// TIA Portal V21 export
FUNCTION_BLOCK "FB304"   // FB304, LAD
TITLE = FB304
{ S7_Optimized_Access := 'TRUE' }
AUTHOR : PRECISE
FAMILY : PRECISE
// BLANKETING
// stored: AutoNumber false, MemoryReserve 100, SetENOAutomatically false
   VAR_INPUT
      Enable : Bool;
      Disable : Bool;
      Fault : Bool;
      SecPulse : Bool;
      AlwaysTrue : Bool;
      StartConfirmationPopupSel : Bool;   // StartConfirmationPopupSel: 0-NO/1-YES
      EndConfirmationPopupSel : Bool;   // EndConfirmationPopupSel: 0-NO/1-YES
      BlanketingModeSel : Int;   // Blanketing Mode Selection: 0-Pressure/1-Pressure+Time
      BlanketingTimebaseSel : Bool;   // Blanketing Timebase Selection: 0-sec/1-min
      GasSel : Int;   // Gas Selection - 0-AIR/1-N2
      SetPressure : Real := 1.0;   // For Blanketing Mode Selection: 0-Pressure
      BlanketingTimeMin : Int := 1;   // For Blanketing Mode Selection: 1-Pressure+Time & Blanketing Timebase Selection: 1-min
      BlanketingTimeSec : Int := 30;   // For Blanketing Mode Selection: 1-Pressure+Time & Blanketing Timebase Selection: 0-sec
      ActualPressure : Real;   // For Sparging LineSelection: 1-THRU VV
      DelaytoOpenGasIn : Int := 3;
      PressureTol : Real := 0.3;
   END_VAR
   VAR_OUTPUT
      AirValve : Bool;
      N2Valve : Bool;
      BlanketingLineValves : Bool;
      StartConfirmationPopup : Bool;   // For Start Confirmation Popup Selection: Yes
      EndConfirmationPopup : Bool;   // For End Confirmation Popup Selection: Yes
      BlanketingTimeMinPV : DInt;
      BlanketingTimeSecPV : DInt;
      PrintTrigger : Bool;
      PrintWord : Int;
      PrintStatus : String[50];
   END_VAR
   VAR_IN_OUT
      Start : Bool;
      Stop : Bool;
      Reset : Bool;
      StartConfirmationAck : Bool;   // For Start Confirmation Popup Selection: Yes
      EndConfirmationAck : Bool;   // For End Confirmation Popup Selection: Yes
      SpareBtn1 : Bool;
      SpareBtn2 : Bool;
      SpareBtn3 : Bool;
      Running : Bool;
      Selected : Bool;
      Paused : Bool;
      StartConfirmationPopupTemp : Bool;   // For Start Confirmation Popup Selection: Yes
      EndConfirmationPopupTemp : Bool;   // For End Confirmation Popup Selection: Yes
      BlanketingStarted : Bool;
      BlanketingOver : Bool;
      BlanketingTimerRunning : Bool;
      PressureTolNeg : Real;
   END_VAR
   VAR
      ValveOnDelayPV : Int;
      ValveOffDelayPV : Int;
      PrintTriggerTemp : Bool;
      RE1 : Bool;
      RE2 : Bool;
      RE3 : Bool;
      RE4 : Bool;
      RE5 : Bool;
      RE6 : Bool;
      RE7 : Bool;
      BlanketingTimer { S7_SetPoint := 'True'} : "FB101";
      PrintTriggerResetTimer { S7_SetPoint := 'True'} : TON_TIME;
      BtnResetTimer { S7_SetPoint := 'True'} : TON_TIME;
   END_VAR
   VAR_TEMP
      STATUS1 : String[40];
      STATUS2 : String[40];
      STATUS3 : String[40];
      STATUS4 : String[40];
      STATUS5 : String[40];
   END_VAR
   VAR_TEMP   // added for the SCL form of the ladder/FBD networks
      _w1 : Bool;
      _w2 : Bool;
      _w3 : Bool;
      _w4 : Bool;
      _w5 : Bool;
   END_VAR
BEGIN

REGION Network 1: Running
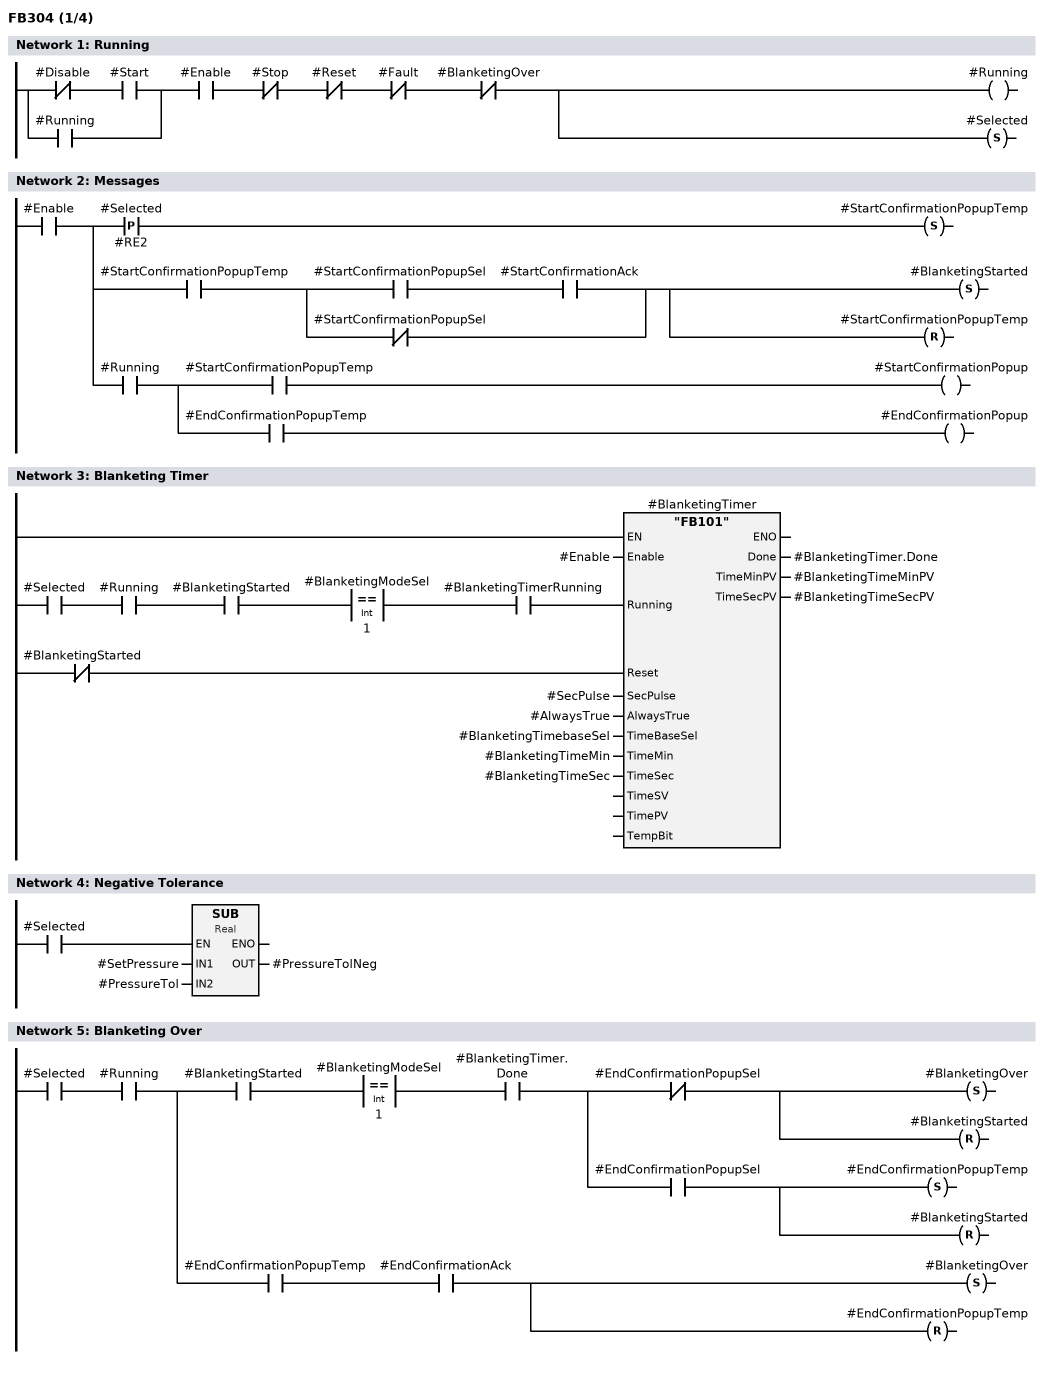
   RUNG wire#powerrail
      I_Contact( #Disable )
      Contact( #Start )
      wire#w1
      Contact( #Enable )
      I_Contact( #Stop )
      I_Contact( #Reset )
      I_Contact( #Fault )
      I_Contact( #BlanketingOver )
      wire#w2
      Coil( #Running )
   END_RUNG
   RUNG wire#powerrail
      Contact( #Running )
   END_RUNG wire#w1
   RUNG wire#w2
      S_Coil( #Selected )
   END_RUNG
   // the same network as SCL:
   #Running := ((NOT #Disable AND #Start) OR #Running) AND #Enable AND NOT #Stop AND NOT #Reset AND NOT #Fault AND NOT #BlanketingOver;
   IF #Running THEN #Selected := TRUE; END_IF;
END_REGION

REGION Network 2: Messages
   RUNG wire#powerrail
      Contact( #Enable )
      wire#w1
      P_Contact(operand := #Selected, bit := #RE2)
      S_Coil( #StartConfirmationPopupTemp )
   END_RUNG
   RUNG wire#w1
      Contact( #StartConfirmationPopupTemp )
      wire#w2
      Contact( #StartConfirmationPopupSel )
      Contact( #StartConfirmationAck )
      wire#w3
      S_Coil( #BlanketingStarted )
   END_RUNG
   RUNG wire#w2
      I_Contact( #StartConfirmationPopupSel )
   END_RUNG wire#w3
   RUNG wire#w3
      R_Coil( #StartConfirmationPopupTemp )
   END_RUNG
   RUNG wire#w1
      Contact( #Running )
      wire#w4
      Contact( #StartConfirmationPopupTemp )
      Coil( #StartConfirmationPopup )
   END_RUNG
   RUNG wire#w4
      Contact( #EndConfirmationPopupTemp )
      Coil( #EndConfirmationPopup )
   END_RUNG
   // the same network as SCL:
   #_w1 := #Enable AND #Selected AND NOT #RE2;   // rising edge of #Selected
   #RE2 := #Selected;
   IF #_w1 THEN #StartConfirmationPopupTemp := TRUE; END_IF;
   IF #Enable AND #StartConfirmationPopupTemp AND ((#StartConfirmationPopupSel AND #StartConfirmationAck) OR NOT #StartConfirmationPopupSel) THEN
       #BlanketingStarted := TRUE;
       #StartConfirmationPopupTemp := FALSE;
   END_IF;
   #_w2 := #Enable AND #Running;
   #StartConfirmationPopup := #_w2 AND #StartConfirmationPopupTemp;
   #EndConfirmationPopup := #_w2 AND #EndConfirmationPopupTemp;
END_REGION

REGION Network 3: Blanketing Timer
   RUNG wire#powerrail
      #BlanketingTimer(Running := wire#w1, Reset := wire#w2, Enable := #Enable, SecPulse := #SecPulse, AlwaysTrue := #AlwaysTrue, TimeBaseSel := #BlanketingTimebaseSel, TimeMin := #BlanketingTimeMin, TimeSec := #BlanketingTimeSec, TimeSV :=, TimePV :=, TempBit :=, Done => #BlanketingTimer.Done, TimeMinPV => #BlanketingTimeMinPV, TimeSecPV => #BlanketingTimeSecPV)
   END_RUNG
   RUNG wire#powerrail
      Contact( #Selected )
      Contact( #Running )
      Contact( #BlanketingStarted )
      { S7_Templates := "SrcType := Int" } EQ_Contact(in1 := #BlanketingModeSel, in2 := 1)
      Contact( #BlanketingTimerRunning )
   END_RUNG wire#w1
   RUNG wire#powerrail
      I_Contact( #BlanketingStarted )
   END_RUNG wire#w2
   // the same network as SCL:
   #BlanketingTimer(Enable := #Enable,   // "FB101"
                    Running := #Selected AND #Running AND #BlanketingStarted AND (#BlanketingModeSel = 1) AND #BlanketingTimerRunning,
                    Reset := NOT #BlanketingStarted,
                    SecPulse := #SecPulse,
                    AlwaysTrue := #AlwaysTrue,
                    TimeBaseSel := #BlanketingTimebaseSel,
                    TimeMin := #BlanketingTimeMin,
                    TimeSec := #BlanketingTimeSec,
                    Done => #BlanketingTimer.Done,
                    TimeMinPV => #BlanketingTimeMinPV,
                    TimeSecPV => #BlanketingTimeSecPV);
END_REGION

REGION Network 4: Negative Tolerance
   RUNG wire#powerrail
      Contact( #Selected )
      { S7_Templates := "SrcType := Real"; S7_GenerateENO := "TRUE" } Sub(in1 := #SetPressure, in2 := #PressureTol, out => #PressureTolNeg)
   END_RUNG
   // the same network as SCL:
   IF #Selected THEN #PressureTolNeg := #SetPressure - #PressureTol; END_IF;
END_REGION

REGION Network 5: Blanketing Over
   RUNG wire#powerrail
      Contact( #Selected )
      Contact( #Running )
      wire#w1
      Contact( #BlanketingStarted )
      { S7_Templates := "SrcType := Int" } EQ_Contact(in1 := #BlanketingModeSel, in2 := 1)
      Contact( #BlanketingTimer.Done )
      wire#w2
      I_Contact( #EndConfirmationPopupSel )
      wire#w3
      S_Coil( #BlanketingOver )
   END_RUNG
   RUNG wire#w3
      R_Coil( #BlanketingStarted )
   END_RUNG
   RUNG wire#w2
      Contact( #EndConfirmationPopupSel )
      wire#w4
      S_Coil( #EndConfirmationPopupTemp )
   END_RUNG
   RUNG wire#w4
      R_Coil( #BlanketingStarted )
   END_RUNG
   RUNG wire#w1
      Contact( #EndConfirmationPopupTemp )
      Contact( #EndConfirmationAck )
      wire#w5
      S_Coil( #BlanketingOver )
   END_RUNG
   RUNG wire#w5
      R_Coil( #EndConfirmationPopupTemp )
   END_RUNG
   // the same network as SCL:
   #_w1 := #Selected AND #Running;
   #_w2 := #_w1 AND #BlanketingStarted AND (#BlanketingModeSel = 1) AND #BlanketingTimer.Done;
   IF #_w2 AND NOT #EndConfirmationPopupSel THEN
       #BlanketingOver := TRUE;
       #BlanketingStarted := FALSE;
   END_IF;
   IF #_w2 AND #EndConfirmationPopupSel THEN
       #EndConfirmationPopupTemp := TRUE;
       #BlanketingStarted := FALSE;
   END_IF;
   IF #_w1 AND #EndConfirmationPopupTemp AND #EndConfirmationAck THEN
       #BlanketingOver := TRUE;
       #EndConfirmationPopupTemp := FALSE;
   END_IF;
END_REGION

REGION Network 6: Output On
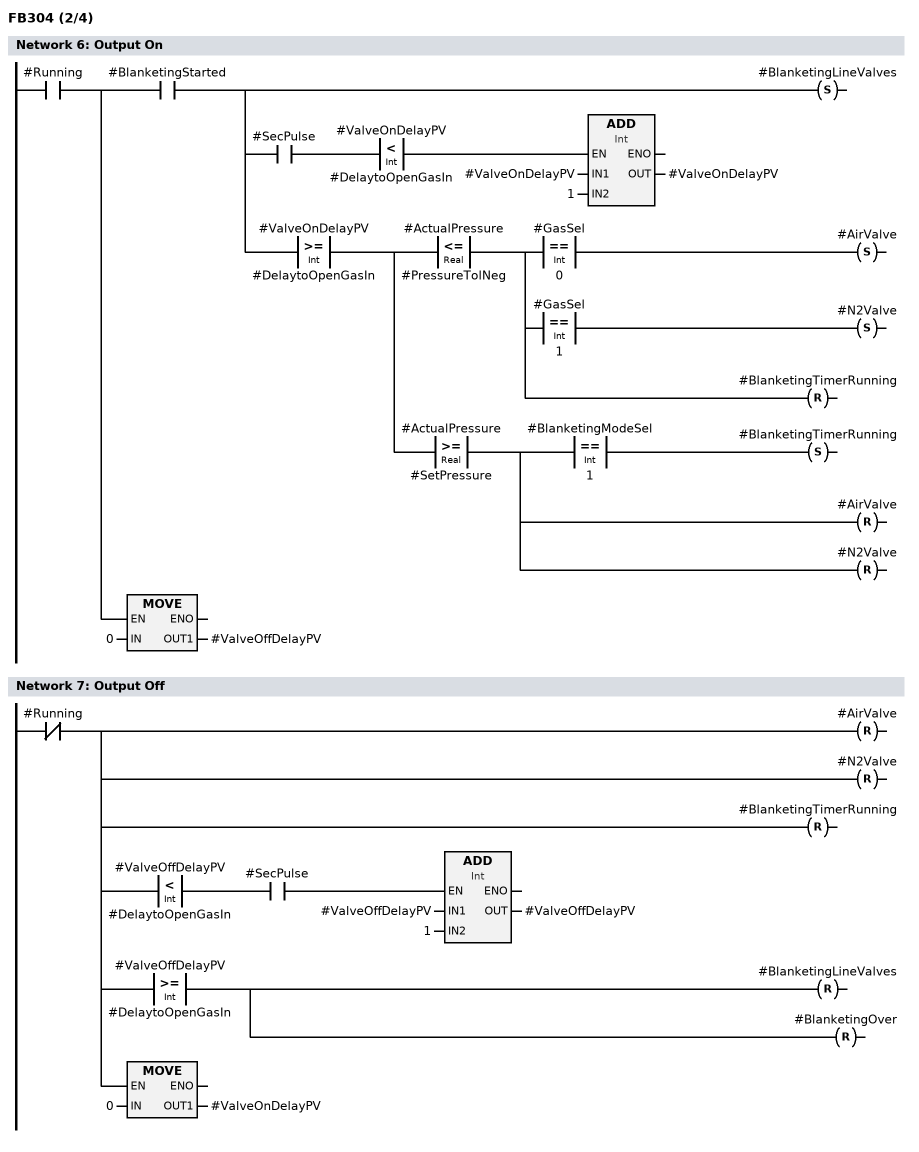
   RUNG wire#powerrail
      Contact( #Running )
      wire#w1
      Contact( #BlanketingStarted )
      wire#w2
      S_Coil( #BlanketingLineValves )
   END_RUNG
   RUNG wire#w2
      Contact( #SecPulse )
      { S7_Templates := "SrcType := Int" } LT_Contact(in1 := #ValveOnDelayPV, in2 := #DelaytoOpenGasIn)
      { S7_Templates := "SrcType := Int"; S7_GenerateENO := "TRUE" } Add(in1 := #ValveOnDelayPV, in2 := 1, out => #ValveOnDelayPV)
   END_RUNG
   RUNG wire#w2
      { S7_Templates := "SrcType := Int" } GE_Contact(in1 := #ValveOnDelayPV, in2 := #DelaytoOpenGasIn)
      wire#w3
      { S7_Templates := "SrcType := Real" } LE_Contact(in1 := #ActualPressure, in2 := #PressureTolNeg)
      wire#w4
      { S7_Templates := "SrcType := Int" } EQ_Contact(in1 := #GasSel, in2 := 0)
      S_Coil( #AirValve )
   END_RUNG
   RUNG wire#w4
      { S7_Templates := "SrcType := Int" } EQ_Contact(in1 := #GasSel, in2 := 1)
      S_Coil( #N2Valve )
   END_RUNG
   RUNG wire#w4
      R_Coil( #BlanketingTimerRunning )
   END_RUNG
   RUNG wire#w3
      { S7_Templates := "SrcType := Real" } GE_Contact(in1 := #ActualPressure, in2 := #SetPressure)
      wire#w5
      { S7_Templates := "SrcType := Int" } EQ_Contact(in1 := #BlanketingModeSel, in2 := 1)
      S_Coil( #BlanketingTimerRunning )
   END_RUNG
   RUNG wire#w5
      R_Coil( #AirValve )
   END_RUNG
   RUNG wire#w5
      R_Coil( #N2Valve )
   END_RUNG
   RUNG wire#w1
      { S7_GenerateENO := "TRUE" } Move(in := 0, out1 => #ValveOffDelayPV)
   END_RUNG
   // the same network as SCL:
   #_w1 := #Running AND #BlanketingStarted;
   IF #_w1 THEN #BlanketingLineValves := TRUE; END_IF;
   IF #_w1 AND #SecPulse AND (#ValveOnDelayPV < #DelaytoOpenGasIn) THEN
       #ValveOnDelayPV := #ValveOnDelayPV + 1;
   END_IF;
   #_w2 := #_w1 AND (#ValveOnDelayPV >= #DelaytoOpenGasIn);
   #_w3 := #_w2 AND (#ActualPressure <= #PressureTolNeg);
   IF #_w3 AND (#GasSel = 0) THEN #AirValve := TRUE; END_IF;
   IF #_w3 AND (#GasSel = 1) THEN #N2Valve := TRUE; END_IF;
   IF #_w3 THEN #BlanketingTimerRunning := FALSE; END_IF;
   #_w4 := #_w2 AND (#ActualPressure >= #SetPressure);
   IF #_w4 AND (#BlanketingModeSel = 1) THEN #BlanketingTimerRunning := TRUE; END_IF;
   IF #_w4 THEN
       #AirValve := FALSE;
       #N2Valve := FALSE;
   END_IF;
   IF #Running THEN #ValveOffDelayPV := 0; END_IF;
END_REGION

REGION Network 7: Output Off
   RUNG wire#powerrail
      I_Contact( #Running )
      wire#w1
      R_Coil( #AirValve )
   END_RUNG
   RUNG wire#w1
      R_Coil( #N2Valve )
   END_RUNG
   RUNG wire#w1
      R_Coil( #BlanketingTimerRunning )
   END_RUNG
   RUNG wire#w1
      { S7_Templates := "SrcType := Int" } LT_Contact(in1 := #ValveOffDelayPV, in2 := #DelaytoOpenGasIn)
      Contact( #SecPulse )
      { S7_Templates := "SrcType := Int"; S7_GenerateENO := "TRUE" } Add(in1 := #ValveOffDelayPV, in2 := 1, out => #ValveOffDelayPV)
   END_RUNG
   RUNG wire#w1
      { S7_Templates := "SrcType := Int" } GE_Contact(in1 := #ValveOffDelayPV, in2 := #DelaytoOpenGasIn)
      wire#w2
      R_Coil( #BlanketingLineValves )
   END_RUNG
   RUNG wire#w2
      R_Coil( #BlanketingOver )
   END_RUNG
   RUNG wire#w1
      { S7_GenerateENO := "TRUE" } Move(in := 0, out1 => #ValveOnDelayPV)
   END_RUNG
   // the same network as SCL:
   IF NOT #Running THEN
       #AirValve := FALSE;
       #N2Valve := FALSE;
       #BlanketingTimerRunning := FALSE;
   END_IF;
   IF NOT #Running AND (#ValveOffDelayPV < #DelaytoOpenGasIn) AND #SecPulse THEN
       #ValveOffDelayPV := #ValveOffDelayPV + 1;
   END_IF;
   IF NOT #Running AND (#ValveOffDelayPV >= #DelaytoOpenGasIn) THEN
       #BlanketingLineValves := FALSE;
       #BlanketingOver := FALSE;
   END_IF;
   IF NOT #Running THEN #ValveOnDelayPV := 0; END_IF;
END_REGION

REGION Network 8: Event Status
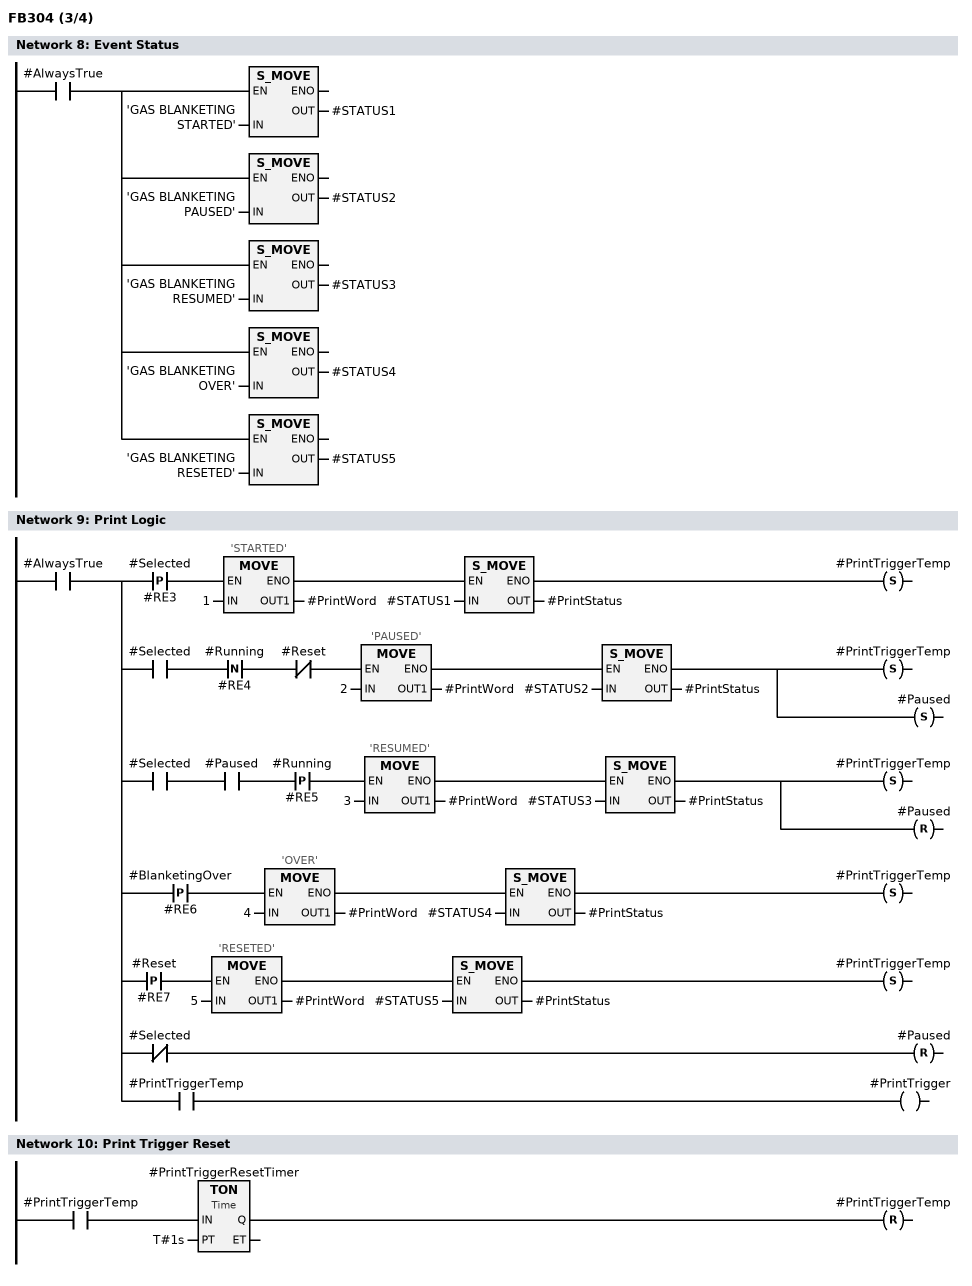
   RUNG wire#powerrail
      Contact( #AlwaysTrue )
      wire#w1
      S_Move(in := 'GAS BLANKETING STARTED', out => #STATUS1)
   END_RUNG
   RUNG wire#w1
      S_Move(in := 'GAS BLANKETING PAUSED', out => #STATUS2)
   END_RUNG
   RUNG wire#w1
      S_Move(in := 'GAS BLANKETING RESUMED', out => #STATUS3)
   END_RUNG
   RUNG wire#w1
      S_Move(in := 'GAS BLANKETING OVER', out => #STATUS4)
   END_RUNG
   RUNG wire#w1
      S_Move(in := 'GAS BLANKETING RESETED', out => #STATUS5)
   END_RUNG
   // the same network as SCL:
   IF #AlwaysTrue THEN
       #STATUS1 := 'GAS BLANKETING STARTED';
       #STATUS2 := 'GAS BLANKETING PAUSED';
       #STATUS3 := 'GAS BLANKETING RESUMED';
       #STATUS4 := 'GAS BLANKETING OVER';
       #STATUS5 := 'GAS BLANKETING RESETED';
   END_IF;
END_REGION

REGION Network 9: Print Logic
   RUNG wire#powerrail
      Contact( #AlwaysTrue )
      wire#w1
      P_Contact(operand := #Selected, bit := #RE3)
      { S7_GenerateENO := "TRUE" } Move(in := 1, out1 => #PrintWord)   // 'STARTED'
      S_Move(in := #STATUS1, out => #PrintStatus)
      S_Coil( #PrintTriggerTemp )
   END_RUNG
   RUNG wire#w1
      Contact( #Selected )
      N_Contact(operand := #Running, bit := #RE4)
      I_Contact( #Reset )
      { S7_GenerateENO := "TRUE" } Move(in := 2, out1 => #PrintWord)   // 'PAUSED'
      S_Move(in := #STATUS2, out => #PrintStatus)
      wire#w2
      S_Coil( #PrintTriggerTemp )
   END_RUNG
   RUNG wire#w2
      S_Coil( #Paused )
   END_RUNG
   RUNG wire#w1
      Contact( #Selected )
      Contact( #Paused )
      P_Contact(operand := #Running, bit := #RE5)
      { S7_GenerateENO := "TRUE" } Move(in := 3, out1 => #PrintWord)   // 'RESUMED'
      S_Move(in := #STATUS3, out => #PrintStatus)
      wire#w3
      S_Coil( #PrintTriggerTemp )
   END_RUNG
   RUNG wire#w3
      R_Coil( #Paused )
   END_RUNG
   RUNG wire#w1
      P_Contact(operand := #BlanketingOver, bit := #RE6)
      { S7_GenerateENO := "TRUE" } Move(in := 4, out1 => #PrintWord)   // 'OVER'
      S_Move(in := #STATUS4, out => #PrintStatus)
      S_Coil( #PrintTriggerTemp )
   END_RUNG
   RUNG wire#w1
      P_Contact(operand := #Reset, bit := #RE7)
      { S7_GenerateENO := "TRUE" } Move(in := 5, out1 => #PrintWord)   // 'RESETED'
      S_Move(in := #STATUS5, out => #PrintStatus)
      S_Coil( #PrintTriggerTemp )
   END_RUNG
   RUNG wire#w1
      I_Contact( #Selected )
      R_Coil( #Paused )
   END_RUNG
   RUNG wire#w1
      Contact( #PrintTriggerTemp )
      Coil( #PrintTrigger )
   END_RUNG
   // the same network as SCL:
   // ENO of a box is taken as its EN; it also drops when the box reports an error
   #_w1 := #AlwaysTrue AND #Selected AND NOT #RE3;   // rising edge of #Selected
   #RE3 := #Selected;
   IF #_w1 THEN
       #PrintWord := 1;   // 'STARTED'
       #PrintStatus := #STATUS1;
       #PrintTriggerTemp := TRUE;
   END_IF;
   #_w2 := #AlwaysTrue AND #Selected AND NOT #Running AND #RE4;   // falling edge of #Running
   #RE4 := #Running;
   IF #_w2 AND NOT #Reset THEN
       #PrintWord := 2;   // 'PAUSED'
       #PrintStatus := #STATUS2;
       #PrintTriggerTemp := TRUE;
       #Paused := TRUE;
   END_IF;
   #_w3 := #AlwaysTrue AND #Selected AND #Paused AND #Running AND NOT #RE5;   // rising edge of #Running
   #RE5 := #Running;
   IF #_w3 THEN
       #PrintWord := 3;   // 'RESUMED'
       #PrintStatus := #STATUS3;
       #PrintTriggerTemp := TRUE;
       #Paused := FALSE;
   END_IF;
   #_w4 := #AlwaysTrue AND #BlanketingOver AND NOT #RE6;   // rising edge of #BlanketingOver
   #RE6 := #BlanketingOver;
   IF #_w4 THEN
       #PrintWord := 4;   // 'OVER'
       #PrintStatus := #STATUS4;
       #PrintTriggerTemp := TRUE;
   END_IF;
   #_w5 := #AlwaysTrue AND #Reset AND NOT #RE7;   // rising edge of #Reset
   #RE7 := #Reset;
   IF #_w5 THEN
       #PrintWord := 5;   // 'RESETED'
       #PrintStatus := #STATUS5;
       #PrintTriggerTemp := TRUE;
   END_IF;
   IF #AlwaysTrue AND NOT #Selected THEN #Paused := FALSE; END_IF;
   #PrintTrigger := #AlwaysTrue AND #PrintTriggerTemp;
END_REGION

REGION Network 10: Print Trigger Reset
   RUNG wire#powerrail
      Contact( #PrintTriggerTemp )
      { S7_Templates := "time_type := Time" } #PrintTriggerResetTimer.TON(pt := T#1s, et =>)
      R_Coil( #PrintTriggerTemp )
   END_RUNG
   // the same network as SCL:
   #PrintTriggerResetTimer(IN := #PrintTriggerTemp, PT := T#1s);   // TON
   IF #PrintTriggerResetTimer.Q THEN #PrintTriggerTemp := FALSE; END_IF;
END_REGION

REGION Network 11: Button Reset
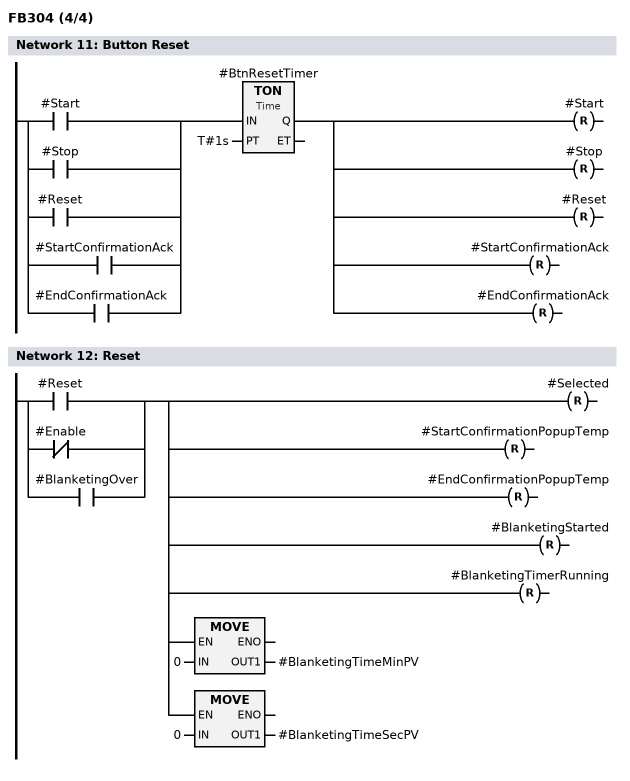
   RUNG wire#powerrail
      Contact( #Start )
      wire#w1
      { S7_Templates := "time_type := Time" } #BtnResetTimer.TON(pt := T#1s, et =>)
      wire#w2
      R_Coil( #Start )
   END_RUNG
   RUNG wire#powerrail
      Contact( #Stop )
   END_RUNG wire#w1
   RUNG wire#powerrail
      Contact( #Reset )
   END_RUNG wire#w1
   RUNG wire#powerrail
      Contact( #StartConfirmationAck )
   END_RUNG wire#w1
   RUNG wire#powerrail
      Contact( #EndConfirmationAck )
   END_RUNG wire#w1
   RUNG wire#w2
      R_Coil( #Stop )
   END_RUNG
   RUNG wire#w2
      R_Coil( #Reset )
   END_RUNG
   RUNG wire#w2
      R_Coil( #StartConfirmationAck )
   END_RUNG
   RUNG wire#w2
      R_Coil( #EndConfirmationAck )
   END_RUNG
   // the same network as SCL:
   #BtnResetTimer(IN := #Start OR #Stop OR #Reset OR #StartConfirmationAck OR #EndConfirmationAck, PT := T#1s);   // TON
   IF #BtnResetTimer.Q THEN
       #Start := FALSE;
       #Stop := FALSE;
       #Reset := FALSE;
       #StartConfirmationAck := FALSE;
       #EndConfirmationAck := FALSE;
   END_IF;
END_REGION

REGION Network 12: Reset
   RUNG wire#powerrail
      Contact( #Reset )
      wire#w1
      R_Coil( #Selected )
   END_RUNG
   RUNG wire#powerrail
      I_Contact( #Enable )
   END_RUNG wire#w1
   RUNG wire#powerrail
      Contact( #BlanketingOver )
   END_RUNG wire#w1
   RUNG wire#w1
      R_Coil( #StartConfirmationPopupTemp )
   END_RUNG
   RUNG wire#w1
      R_Coil( #EndConfirmationPopupTemp )
   END_RUNG
   RUNG wire#w1
      R_Coil( #BlanketingStarted )
   END_RUNG
   RUNG wire#w1
      R_Coil( #BlanketingTimerRunning )
   END_RUNG
   RUNG wire#w1
      { S7_GenerateENO := "TRUE" } Move(in := 0, out1 => #BlanketingTimeMinPV)
   END_RUNG
   RUNG wire#w1
      { S7_GenerateENO := "TRUE" } Move(in := 0, out1 => #BlanketingTimeSecPV)
   END_RUNG
   // the same network as SCL:
   IF #Reset OR NOT #Enable OR #BlanketingOver THEN
       #Selected := FALSE;
       #StartConfirmationPopupTemp := FALSE;
       #EndConfirmationPopupTemp := FALSE;
       #BlanketingStarted := FALSE;
       #BlanketingTimerRunning := FALSE;
       #BlanketingTimeMinPV := 0;
       #BlanketingTimeSecPV := 0;
   END_IF;
END_REGION
END_FUNCTION_BLOCK
